FUNCTION setEventInfo : BOOL
VAR_INPUT
	events				: REFERENCE TO ST_Events;
	stEvent 			: REFERENCE TO ST_Event;
	isError				: BOOL;
	strMessage 			: STRING(255);
END_VAR

stEvent.message := strMessage;
stEvent.isTriggered := TRUE;
updateEventWithTimestamp(stEvent := stEvent);
events.errorsDetected := isError;

END_FUNCTION

(* stored: Version 1.1.0.1
   POU setEventInfo: Id {fd5c5f94-c786-40c8-961b-6509209e48e8}, SpecialFunc None *)
